# EPICS alarm handler configuration: epics/epics_alh/alarms_list_TargetDAQ.alhConfig
GROUP NULL TargetDAQ
